FUNCTION_BLOCK FB_TIIAlarmDbStn
VAR_INPUT
	vIO 					: ST_DebugStation_VIO;
	NoOfTIIAlm 				: INT	:= NO_OF_TII_SENSOR;
	iLevel 					: INT	:= 1;
END_VAR
VAR_OUTPUT
	isTIIError				: BOOL;
	TIIAlarmLED					: BOOL;
END_VAR
VAR
	DIFU					: R_TRIG;
	tim 					: TON;
	delay 					: FB_Delay;
	tPOn					: BOOL;	//testerPowerOutoutOn after Delay
	dPOn					: BOOL; //dpsPwrbit after Delay
	bitNo					: INT;
	alarmReset				: BOOL;
	
	ArrAlmBitBefDelay 		: ARRAY[1..NO_OF_TII_SENSOR] OF BOOL;
	ArrAlmBitAftDelay 		: ARRAY[1..NO_OF_TII_SENSOR] OF BOOL;
	ArrAlarmKeepBit			: ARRAY[1..NO_OF_TII_SENSOR] OF BOOL;
	ArrDelayAlarm 			: ARRAY[1..NO_OF_TII_SENSOR] OF FB_AlarmDelay;
	Arr_ms 					: ARRAY[1..NO_OF_TII_SENSOR] OF INT;
	bTIIByPassArray			: ARRAY[1..NO_OF_TII_SENSOR] OF BOOL;
	i						: INT;
	bTest 					: BOOL;
END_VAR

//<HMI_TII_Test>

	IF bHMITIIBypass THEN
		bTIIByPassArray:= stHMITIIByPassArray[iLevel].bHMITIIByPassArray;
		//FOR i:=1 TO NoOfTIIAlm DO
		//	bTIIByPassArray[i]:= NOT stHMITIIByPassArray[iLevel].bHMITIIByPassArray[i];
		//END_FOR
	ELSE
		FOR i:=1 TO NoOfTIIAlm DO
			//bTIIByPassArray[i]:=bEnableTIIAlarm;
			bTIIByPassArray[i]:=TC_ModuleState[iLevel].TCSite[1].TIERII = E_State.eEnabled;
		END_FOR
	END_IF
//</HMI_TII_Test>
//IF bTest THEN
AlarmUpdate(bENs:=bTIIByPassArray);
//END_IF

METHOD AlarmUpdate : BOOL
VAR
	i						: INT;
	j						: INT;
	_bError					: BOOL;
	iSysAlarmID 			: INT;
	e						: E_TIIAlarm;
	bTstOnCmd 				: BOOL;
	bChkTstOn 				: BOOL;
	
	bAPOnCmd				: BOOL;
	bChkAPOn 				: BOOL;
	//Condition
	lRt:BOOL;
	lEt:BOOL;;
END_VAR

VAR_INPUT
	bENs :ARRAY[1..NO_OF_TII_SENSOR] OF BOOL;
END_VAR

VAR_IN_OUT
	//ArrAlarmKeepBit:ST_AlarmTags;
END_VAR
VAR_OUTPUT
END_VAR
IF iLevel=0 THEN
	RETURN;
END_IF

FOR i:=1 TO NoOfTIIAlm DO	
	CASE i OF
        E_TIIAlarm.ipAPPowerOn: 
			e															:= E_TIIAlarm.ipAPPowerOn; 
			ArrAlmBitBefDelay[E_TIIAlarm.ipAPPowerOn]					:= (NOT vIO.ipDBStnAPPowerOn) AND VIO.ipDBStnAPPresentSensor AND GVL_DUT_DC_AP240ACPower.Failed AND bENs[2];
			Arr_ms[e] 													:= 500;  (*TIIAlmText[e]:='AP_PowerOn'*); 
			
	    E_TIIAlarm.ipAPReady: 
			e															:= E_TIIAlarm.ipAPReady; 
			ArrAlmBitBefDelay[E_TIIAlarm.ipAPReady]						:= (NOT	vIO.ipDBStnAPReady)	AND vIO.ipDBStnAPPresentSensor AND bENs[3]; 	
			Arr_ms[e] 													:= 500;  (*TIIAlmText[e]:='AP_Ready' 		    	*);     
                   
	    E_TIIAlarm.ipCellGroundFault:
			e															:= E_TIIAlarm.ipCellGroundFault; 
			ArrAlmBitBefDelay[E_TIIAlarm.ipCellGroundFault]				:= vIO.ipDBStnCellGroundFault AND bENs[8] ; 
			Arr_ms[e] 													:= 500;  //TIIAlmText[e]:='CellGroundFault'  		;    

		E_TIIAlarm.ipCellFluidLeakage1: 
			e															:= E_TIIAlarm.ipCellFluidLeakage1; 
			ArrAlmBitBefDelay[E_TIIAlarm.ipCellFluidLeakage1]			:= vIO.ipDBStnCellFluidLeakage1 (*AND bENs[6]*); 			
			Arr_ms[e] 													:= 500;  (*TIIAlmText[e]:='CellFluidLeakage1' 	*);   
			
	    E_TIIAlarm.ipCellFluidLeakage2: 
			e															:= E_TIIAlarm.ipCellFluidLeakage2; 
			ArrAlmBitBefDelay[E_TIIAlarm.ipCellFluidLeakage2]			:= vIO.ipDBStnCellFluidLeakage2 (*AND bENs[7]*) ; 			
			Arr_ms[e] 													:= 500;  (*TIIAlmText[e]:='CellFluidLeakage2'*);     
	END_CASE

	//Delay Library Alm Bit
	ArrDelayAlarm[i](	alarmState			:= ArrAlmBitBefDelay[i],
						triggerAlarmState	=> ArrAlmBitAftDelay[i],
						alarmResetTimer		:= alarmReset,
						msec				:= Arr_ms[i]);	//DelayAlmBit
	

	IF ArrAlmBitAftDelay[i] THEN					//realtime IO update array
		//stAlmMod.Level[iLevel].AlarmID[i]:=TRUE;
		ALMTC.Level[iLevel].AlarmID[i]:=TRUE;
	ELSE
		//TIIAlmText[i]:='';  
	END_IF		
		//_bError := _bError OR stAlmMod.Level[iLevel].AlarmID[i];
		_bError := _bError OR ALMTC.Level[iLevel].AlarmID[i];
	
END_FOR

TIIAlarmLED															:=		ALMTC.Level[iLevel].AlarmID[E_TIIAlarm.ipAPPowerOn 		   	   		]   OR 
		    																ALMTC.Level[iLevel].AlarmID[E_TIIAlarm.ipAPReady		       	   	]   OR
																			ALMTC.Level[iLevel].AlarmID[E_TIIAlarm.ipCellFluidLeakage1		   	]   OR
																			ALMTC.Level[iLevel].AlarmID[E_TIIAlarm.ipCellFluidLeakage2		   	]   OR
																			ALMTC.Level[iLevel].AlarmID[E_TIIAlarm.ipCellGroundFault 	   		];
END_METHOD

PROPERTY P_ErrClear : BOOL
GET
END_GET
SET
alarmReset	:= P_ErrClear;
END_SET
END_PROPERTY

END_FUNCTION_BLOCK

(* stored: Version 1.1.0.1, ProductVersion 3.1.4022.18
   POU FB_TIIAlarmDbStn: Id {1f1c0a9a-a15d-4901-bcd2-0649d00aa61a}, SpecialFunc None
   Method AlarmUpdate: Id {df4f023a-29b0-4ee7-baee-77dc81ad8f78}
   Property P_ErrClear: Id {400cb5c4-2dc6-4fab-b5e3-d1a6a6655309}
   Get Get: Id {e7f3b0b1-d5ff-4651-92e7-f2b82d74132a}
   Set Set: Id {ecaf4f2d-d579-4242-ac6c-78cd914d372d} *)
